  ft_insert_part_state=0
  ft_insert_part_return=0
  ft_sensor_filter_insertpart_hex=6
  ft_insert_part_frameID=1
  ft_insert_part_frameID_default=1
  ft_insert_part_frameRPY=ON_ZERO3D
  ft_insert_part_frameRPY_default=ON_ZERO3D
  ft_insert_part_retAccept=[True,True,True,False,False,False,False,False,False]
  ft_insert_part_retAccept_default=[True,True,True,False,False,False,False,False,False]
  FT_INSERT_PART_STATE_IDLE=0
  FT_INSERT_PART_STATE_INIT=1
  FT_INSERT_PART_STATE_STARTED=2
  FT_INSERT_PART_STATE_RETURNING=3
  ft__insert_part_param_error_minDistZ="Please define parameter 'minDistZ' as a positive real number in meters!"
  ft__insert_part_param_error_forceZ="Please define parameter 'forceZ' as a positive number in Newtons!"
  ft__insert_part_param_error_maxDistZ="Please define parameter 'maxDistZ' as a positive real number in meters!"
  ft__insert_part_param_error_maxDistZ_minDistZ="Please define the parameters as 'maxDistZ' >= 'minDistZ'!"
  ft__insert_part_param_error_expSpeed="Please define parameter 'expSpeed' as a positive real number in meters!"
  ft__insert_part_param_error_deltaForce="Please define parameter 'deltaForce' as a positive number in Newtons!"
  ft__insert_part_param_error_timeOut="Please define parameter 'timeOut' as a positive number in seconds!"
  ft__insert_part_param_error_FTLimits="Please define parameter 'FTLimits' as a 6-element array of positive numbers in Newtons & Newton-meters!"
  ft__insert_part_param_error_PGainFxy="Please define parameter 'PGainFxy' as a positive real number!"
  ft__insert_part_param_error_PGainFz="Please define parameter 'PGainFz' as a positive real number!"
  ft__insert_part_param_error_PGainTxy="Please define parameter 'PGainTxy' as a positive real number!"
  ft__insert_part_param_error_PGainTz="Please define parameter 'PGainTz' as a positive real number!"
  def ft_insert_part(forceZ,minDistZ,maxDistZ=0.0,deltaForce=0.0,expSpeed=0.0,timeOut=0,compliance=[True,True,True,True,True,True],FTLimits=ON_ZERO6D,PGainFxy=1.0,PGainFz=1.0,PGainTxy=0.2,PGainTz=0.2,popupmsg=True):
  sync()
  if ON_DEBUG_LOG:
  textmsg("Insert Part starting..")
  end
  if not(ft_insert_part_state==FT_INSERT_PART_STATE_IDLE):
  textmsg("ft_insert_part_state: ",ft_insert_part_state)
  popup(ft_insert_part_state_error_start,title=ft_insert_part_error_title,error=True,blocking=False)
  halt
  else:
  enter_critical
  ft_insert_part_state=FT_INSERT_PART_STATE_INIT
  exit_critical
  end
  ft_insert_part_return=0
  if not(minDistZ>=0):
  ft_insert_part_return=8
  popup(ft__insert_part_param_error_minDistZ,title=ft_insert_part_error_title,error=True,blocking=True)
  elif not(forceZ!=0):
  ft_insert_part_return=8
  popup(ft__insert_part_param_error_forceZ,title=ft_insert_part_error_title,error=True,blocking=True)
  elif not(maxDistZ>=0):
  ft_insert_part_return=8
  popup(ft__insert_part_param_error_maxDistZ,title=ft_insert_part_error_title,error=True,blocking=False)
  elif not(maxDistZ>=minDistZ or maxDistZ==0):
  ft_insert_part_return=8
  popup(ft__insert_part_param_error_maxDistZ_minDistZ,title=ft_insert_part_error_title,error=True,blocking=False)
  elif not(expSpeed>=0):
  ft_insert_part_return=8
  popup(ft__insert_part_param_error_expSpeed,title=ft_insert_part_error_title,error=True,blocking=False)
  elif not(deltaForce>=0):
  ft_insert_part_return=8
  popup(ft__insert_part_param_error_deltaForce,title=ft_insert_part_error_title,error=True,blocking=False)
  elif not(timeOut>=0):
  ft_insert_part_return=8
  popup(ft__insert_part_param_error_timeOut,title=ft_insert_part_error_title,error=True,blocking=False)
  elif not(FTLimits[0]>=0):
  ft_insert_part_return=8
  popup(ft__insert_part_param_error_FTLimits,title=ft_insert_part_error_title,error=True,blocking=False)
  elif not(FTLimits[1]>=0):
  ft_insert_part_return=8
  popup(ft__insert_part_param_error_FTLimits,title=ft_insert_part_error_title,error=True,blocking=False)
  elif not(FTLimits[3]>=0):
  ft_insert_part_return=8
  popup(ft__insert_part_param_error_FTLimits,title=ft_insert_part_error_title,error=True,blocking=False)
  elif not(FTLimits[4]>=0):
  ft_insert_part_return=8
  popup(ft__insert_part_param_error_FTLimits,title=ft_insert_part_error_title,error=True,blocking=False)
  elif not(FTLimits[5]>=0):
  ft_insert_part_return=8
  popup(ft__insert_part_param_error_FTLimits,title=ft_insert_part_error_title,error=True,blocking=False)
  elif not(PGainFxy>0):
  ft_insert_part_return=8
  popup(ft__insert_part_param_error_PGainFxy,title=ft_insert_part_error_title,error=True,blocking=False)
  elif not(PGainFz>0):
  ft_insert_part_return=8
  popup(ft__insert_part_param_error_PGainFz,title=ft_insert_part_error_title,error=True,blocking=False)
  elif not(PGainTxy>0):
  ft_insert_part_return=8
  popup(ft__insert_part_param_error_PGainTxy,title=ft_insert_part_error_title,error=True,blocking=False)
  elif not(PGainTz>0):
  ft_insert_part_return=8
  popup(ft__insert_part_param_error_PGainTz,title=ft_insert_part_error_title,error=True,blocking=False)
  end
  if(ft_insert_part_return!=0):
  halt
  end
  on_tcp_offset_send(get_tcp_offset())
  local retAccept=ft_insert_part_retAccept
  ft_insert_part_retAccept=ft_insert_part_retAccept_default
  local ft_compliance=compliance
  ft_compliance[2]=True
  local ft_threshold=[FTLimits[0],FTLimits[1],(forceZ+deltaForce),FTLimits[3],FTLimits[4],FTLimits[5]]
  i=0
  while i<6:
  if ft_compliance[i]:
  ft_threshold[i]=0
  end
  i=i+1
  end
  local flags=binary_list_to_integer(ft_compliance)+(ft_insert_part_frameID*64)
  ft_insert_part_frameID=ft_insert_part_frameID_default
  local ft_insert_part_frame=rpy2rotvec(ft_insert_part_frameRPY)
  ft_insert_part_frameRPY=ft_insert_part_frameRPY_default
  sync()
  ft_insert_part_return=ft_pin_insertion(minDistZ,forceZ,compliance,maxDistZ,expSpeed,deltaForce,timeOut,FTLimits,PGainFxy,PGainFz,PGainTxy,PGainTz)
  if ON_DEBUG_LOG:
  textmsg("Insert Part returned.")
  end
  if ft_insert_part_return==0:
  if(popupmsg and(not retAccept[0])):
  popup(ft_insert_part_return_0,title=ft_insert_part_return_title,warning=True,blocking=True)
  end
  elif ft_insert_part_return==1:
  if(popupmsg and(not retAccept[1])):
  popup(ft_insert_part_return_1,title=ft_insert_part_return_title,warning=True,blocking=True)
  end
  elif ft_insert_part_return==2:
  if(popupmsg and(not retAccept[2])):
  popup(ft_insert_part_return_2,title=ft_insert_part_return_title,warning=True,blocking=True)
  end
  elif ft_insert_part_return==3:
  if(popupmsg and(not retAccept[3])):
  popup(ft_insert_part_return_3,title=ft_insert_part_return_title,warning=True,blocking=True)
  end
  elif ft_insert_part_return==4:
  if(popupmsg and(not retAccept[4])):
  popup(ft_insert_part_return_4,title=ft_insert_part_return_title,warning=True,blocking=True)
  end
  elif ft_insert_part_return==5:
  if(popupmsg and(not retAccept[5])):
  popup(ft_insert_part_return_5,title=ft_insert_part_return_title,warning=True,blocking=True)
  end
  elif ft_insert_part_return==6:
  if(popupmsg and(not retAccept[6])):
  popup(ft_insert_part_return_6,title=ft_insert_part_return_title,warning=True,blocking=True)
  end
  elif ft_insert_part_return==7:
  if(popupmsg and(not retAccept[7])):
  popup(ft_insert_part_return_7,title=ft_insert_part_return_title,warning=True,blocking=True)
  end
  else:
  popup(ft_insert_part_return_unknown,title=ft_insert_part_return_title,warning=True,blocking=True)
  end
  enter_critical
  ft_insert_part_state=FT_INSERT_PART_STATE_IDLE
  exit_critical
  if ON_DEBUG_LOG:
  textmsg("End of Insert Part.")
  end
  return ft_insert_part_return
  end
  ft_peakFzScanner_flag=False
  ft_abs_Fz=0
  ft_abs0_Fz=False
  thread ft_peakFzScanner():
  ft_peakFzScanner_flag=True
  ft_abs_Fz=0
  while(ft_peakFzScanner_flag==True):
  local norm_Fz=norm(FT_Tool[2])
  if(ft_abs0_Fz):
  ft_abs_Fz=0
  ft_abs0_Fz=False
  elif(ft_abs_Fz<norm_Fz):
  ft_abs_Fz=norm_Fz
  end
  sync()
  end
  end
  ft_fpid_i_pin=0.0
  ft_fpid_d_pin=0.0
  ft_fpid_i_pin_default=0.0
  ft_fpid_d_pin_default=0.0
  ft_tpid_i_pin=0.0
  ft_tpid_d_pin=0.0
  ft_tpid_i_pin_default=0.0
  ft_tpid_d_pin_default=0.0
  def ft_pin_insertion(minDistZ,forceZ,compliance=[True,True,True,True,True,True],maxDistZ=0,expSpeed=0,deltaForce=1,timeOut=0,FTLimits=[999,999,0,999,999,999],PGainFxy=1.0,PGainFz=1.0,PGainTxy=0.2,PGainTz=0.2):
  sync()
  local pinRet=0
  local frameID=1
  local startPose=get_actual_tcp_pose()
  if maxDistZ==0:
  maxDistZ=minDistZ
  end
  local dist2Reach=maxDistZ
  sync()
  local selectThreshold=[False,False,False,False,False,False]
  local ft_select=compliance
  ft_select[2]=True
  local ft_values=[0.0,0.0,0.0,0.0,0.0,0.0]
  ft_values[2]=forceZ+0.0
  local i=0
  while(i<6):
  selectThreshold[i]=not(ft_select[i])
  i=i+1
  end
  local pin_useTimeOut=True
  if timeOut==0:
  pin_useTimeOut=False
  end
  local timeOut100ms=timeOut*10
  local deltaD=expSpeed/10
  ft_pin_currentDist=0
  local peakScanner=run ft_peakFzScanner()
  sync()
  local pin_gainP=[PGainFxy,PGainFxy,PGainFz,PGainTxy,PGainTxy,PGainTz]
  local pin_gainI=[ft_fpid_i_pin,ft_fpid_i_pin,ft_fpid_i_pin,ft_tpid_i_pin,ft_tpid_i_pin,ft_tpid_i_pin]
  local pin_gainD=[ft_fpid_d_pin,ft_fpid_d_pin,ft_fpid_d_pin,ft_tpid_d_pin,ft_tpid_d_pin,ft_tpid_d_pin]
  if on_hex:
  on_xmlrpc.ft_sensor_filter(ft_sensor_filter_insertpart_hex)
  end
  ft_ftcontrol_start(ft_select=ft_select,ft_values=ft_values,frameID=frameID,frameRPY=[0,0,0],gainP=pin_gainP,gainI=pin_gainI,gainD=pin_gainD)
  local cntr=0
  local leaveInsertion=False
  local bumpZeroPeak=True
  local pin_actual_pose=get_actual_tcp_pose()
  ft_pin_currentDist=point_dist(startPose,pin_actual_pose)
  local pin_last_pose=pin_actual_pose
  ft_actual_deltaD=deltaD
  while((ft_pin_currentDist<dist2Reach)and not leaveInsertion):
  on_wait_ms(100)
  pin_actual_pose=get_actual_tcp_pose()
  ft_pin_currentDist=point_dist(startPose,pin_actual_pose)
  ft_actual_deltaD=(ft_actual_deltaD+pose_dist(pin_last_pose,pin_actual_pose))/2
  if(ft_threshold_check(FTLimits,selectThreshold,True)):
  leaveInsertion=True
  if(ft_pin_currentDist<minDistZ):
  pinRet=7
  else:
  pinRet=6
  end
  ft_ftcontrol_stop()
  elif(pin_useTimeOut and(cntr>timeOut100ms)):
  leaveInsertion=True
  if(ft_pin_currentDist<minDistZ):
  pinRet=5
  else:
  pinRet=4
  end
  ft_ftcontrol_stop()
  elif(ft_actual_deltaD<deltaD and cntr>=10):
  leaveInsertion=True
  if(ft_pin_currentDist<minDistZ):
  pinRet=3
  ft_ftcontrol_stop()
  else:
  pinRet=2
  end
  elif(ft_pin_currentDist>=minDistZ):
  if bumpZeroPeak:
  bumpZeroPeak=False
  ft_abs0_Fz=True
  sync()
  else:
  if(ft_abs_Fz>norm(forceZ+deltaForce)and not ft_abs0_Fz):
  ft_peakFzScanner_flag=False
  leaveInsertion=True
  pinRet=1
  end
  end
  end
  pin_last_pose=pin_actual_pose
  cntr=cntr+1
  sync()
  end
  ft_ftcontrol_stop()
  on_xmlrpc.ft_sensor_filter(ft_sensor_filter)
  ft_peakFzScanner_flag=False
  kill peakScanner
  ft_fpid_i_pin=ft_fpid_i_pin_default
  ft_fpid_d_pin=ft_fpid_d_pin_default
  ft_tpid_i_pin=ft_tpid_i_pin_default
  ft_tpid_d_pin=ft_tpid_d_pin_default
  return pinRet
  end

  #======    End of OnRobot FT Insert Part    ======#

  #======    End of OnRobot RG2-FT Proximity AVG Messages    ======#
  #======    OnRobot RG2-FT Proximity AVG    ======#

  rg2ft_proxi_avg_window_default=10
  rg2ft_proxi_avg_window=10
  rg2ft_proxi_avg_window_last=rg2ft_proxi_avg_window
  rg2ft__proxi_avg_window_error_title="OnRobot - Gripper Proximity"
  rg2ft__proxi_avg_window_error_windowSize="Please define parameter windowSize as a positive integer between 0 and 20."
  def rg2ft_proxi_avg_window_set(windowSize=10):
  sync()
  if ON_DEBUG_LOG:
  textmsg("Gripper Proxi Avg Window Set command starting..")
  end
  windowSize=floor(windowSize+0.5)
  if not(windowSize>0 and windowSize<=20):
  popup(rg2ft__proxi_avg_window_error_windowSize,title=rg2ft__proxi_avg_window_error_title,error=True,blocking=False)
  halt
  end
  rg2ft_proxi_avg_window_last=rg2ft_proxi_avg_window
  rg2ft_proxi_avg_window=windowSize
  on_xmlrpc.rg2ft_proxi_avg(windowSize)
  if ON_DEBUG_LOG:
  textmsg("Gripper Proxi Avg Window Set command ended.")
  end
  end
  def rg2ft_proxi_avg_window_reset_last():
  rg2ft_proxi_avg_window_set(rg2ft_proxi_avg_window_last)
  end
  def rg2ft_proxi_avg_window_reset_default():
  rg2ft_proxi_avg_window_set(rg2ft_proxi_avg_window_default)
  end

  #======    End of OnRobot RG2-FT Proximity AVG    ======#

  #======    End of OnRobot RG2-FT Width Filter Messages    ======#
  #======    OnRobot RG2-FT Width Filter    ======#

  rg2ft_width_filter=10
  rg2ft__width_filter_error_title="OnRobot - Gripper Proximity"
  rg2ft__width_filter_error_bufferSize="Please define parameter bufferSize as a positive integer between 0 and 20."
  def rg2ft_width_filter_set(bufferSize=10):
  sync()
  if ON_DEBUG_LOG:
  textmsg("Gripper Width filtering set command starting..")
  end
  bufferSize=floor(bufferSize+0.5)
  if not(bufferSize>0 and bufferSize<=20):
  popup(rg2ft__width_filter_error_bufferSize,title=rg2ft__width_filter_error_title,error=True,blocking=False)
  halt
  end
  rg2ft_width_filter=bufferSize
  on_xmlrpc.rg2ft_width_filter(bufferSize)
  if ON_DEBUG_LOG:
  textmsg("Gripper Width filtering set command stopping..")
  end
  end

  #======    End of OnRobot RG2-FT Width Filter    ======#
  # end: URCap Installation Node
  while (True):
    $ 1 "Robot Program"
    # begin: URCap Program Node
    #   Source: OnRobot, 5.2.0, OnRobot A/S
    #   Type: RG Grip
    $ 2 "RG Grip"
on_return = rg2ft_grip(99.9, 40.0, tool_index = 0, blocking = True, depth_comp = True, popupmsg = True)
rg2ft_payload_set(mass = 0.0, tool_index = 0, use_guard = True)
    # end: URCap Program Node
    $ 3 "Wait: 1.0"
    sleep(1.0)
    # begin: URCap Program Node
    #   Source: OnRobot, 5.2.0, OnRobot A/S
    #   Type: RG Grip
    $ 4 "RG Grip"
on_return = rg2ft_grip(29.6, 40.0, tool_index = 0, blocking = True, depth_comp = True, popupmsg = True)
rg2ft_payload_set(mass = 0.0, tool_index = 0, use_guard = True)
    # end: URCap Program Node
    $ 5 "Wait: 1.0"
    sleep(1.0)
    # begin: URCap Program Node
    #   Source: OnRobot, 5.2.0, OnRobot A/S
    #   Type: TCP
    $ 6 "TCP"
    on_tcp_set_actual_to(isPrimary = True)
    on_tcp_offset_forced_set_actual(isPrimary = 0)
    # end: URCap Program Node
  end
end
